FUNCTION_BLOCK Five_State_Actuator_CAT_HMI (* Service Interface Function Block Type *)
  (* Standard: 61499-2 *)
  (* Version 0.0, 10/7/2025, Schneider Electric, template *)
  PACKAGE Main;
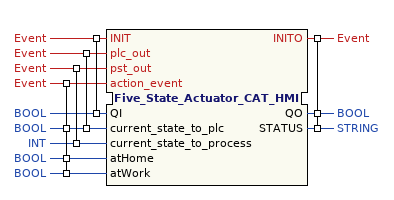
  EVENT_INPUT
    INIT WITH QI;
    plc_out WITH current_state_to_plc;
    pst_out WITH current_state_to_process;
    action_event WITH current_state_to_plc, atHome, atWork;
  END_EVENT
  EVENT_OUTPUT
    INITO WITH QO, STATUS;
  END_EVENT
  VAR_INPUT
    QI : BOOL;
    current_state_to_plc : BOOL;
    current_state_to_process : INT;
    atHome : BOOL;
    atWork : BOOL;
  END_VAR
  VAR_OUTPUT
    QO : BOOL; (* Event Output Qualifier *)
    STATUS : STRING; (* Service Status *)
  END_VAR
  SERVICE /
    SEQUENCE 
    END_SEQUENCE
  END_SERVICE
END_FUNCTION_BLOCK
